// TIA Portal V20 export
FUNCTION_BLOCK "Sequence_1_Cutter"   // FB125, LAD
TITLE = Sequence
// Sequence template programmend in ladder logic
// stored: IsIECCheckEnabled true, MemoryReserve 100, Namespace Unit1.Em4, SetENOAutomatically true
   VAR
      instSequenceLADControl { ExternalWritable := 'False'} : "LAF_ControlLadSequence";
      instSequenceLADStatus { ExternalWritable := 'False'} : "LAF_StatusLadSequence";
      statPulse { ExternalWritable := 'False'} : Array[0..999] of Bool;
      statTonTimer { ExternalWritable := 'False'} : Array[0..999] of TON_TIME;
   END_VAR
   VAR_TEMP
      tempCustomerAction : Bool;   // Placeholder for possible actions
      tempDo_nothing_and_wait_for_init : Bool;   // Placeholder for doing nothing
      tempSafeStateCondition : Bool;   // Temp Condition for the equipment module to be in a safe state
   END_VAR
   VAR CONSTANT
      STEP_IDLE : DInt := 1;   // Idle Step
      JOB_1_STEP_01 : DInt := 101;
      JOB_1_STEP_11 : DInt := 111;
      JOB_1_STEP_21 : DInt := 121;
      JOB_1_STEP_31 : DInt := 131;
      JOB_1_STEP_41 : DInt := 141;
      JOB_1_STEP_51 : DInt := 151;
      JOB_1_STEP_61 : DInt := 161;
      JOB_1_STEP_71 : DInt := 171;
      JOB_1_STEP_81 : DInt := 181;
      JOB_1_STEP_91 : DInt := 191;
      JOB_2_STEP_01 : DInt := 201;
      JOB_2_STEP_11 : DInt := 211;
      JOB_2_STEP_21 : DInt := 221;
      JOB_2_STEP_31 : DInt := 231;
      JOB_2_STEP_41 : DInt := 241;
      JOB_2_STEP_51 : DInt := 251;
      JOB_2_STEP_61 : DInt := 261;
      JOB_2_STEP_71 : DInt := 271;
      JOB_2_STEP_81 : DInt := 281;
      JOB_2_STEP_91 : DInt := 291;
      JOB_3_STEP_01 : DInt := 301;
      JOB_3_STEP_11 : DInt := 311;
      JOB_3_STEP_21 : DInt := 321;
      JOB_3_STEP_31 : DInt := 331;
      JOB_3_STEP_41 : DInt := 341;
      JOB_3_STEP_51 : DInt := 351;
      JOB_3_STEP_61 : DInt := 361;
      JOB_3_STEP_71 : DInt := 371;
      JOB_3_STEP_81 : DInt := 381;
      JOB_3_STEP_91 : DInt := 391;
      JOB_4_STEP_01 : DInt := 401;
      JOB_4_STEP_11 : DInt := 411;
      JOB_4_STEP_21 : DInt := 421;
      JOB_4_STEP_31 : DInt := 431;
      JOB_4_STEP_41 : DInt := 441;
      JOB_4_STEP_51 : DInt := 451;
      JOB_4_STEP_61 : DInt := 461;
      JOB_4_STEP_71 : DInt := 471;
      JOB_4_STEP_81 : DInt := 481;
      JOB_4_STEP_91 : DInt := 491;
      STEP_IMMEDIATE_STOP : DInt := 901;   // Step executed when an immediate stop command is triggered for the sequence (i.e. when unit is in state aborting)
      SeqDelayTime : Time := T#100ms;
      SeqNoDelayTime : Time;
      TRUE : Bool := TRUE;
      FALSE : Bool := FALSE;
      PositionMovingAxisXCuttingPos : SInt := 1;
   END_VAR
   VAR_TEMP   // added for the SCL form of the ladder/FBD networks
      _w1 : Bool;
   END_VAR
BEGIN

REGION Network 1: BLOCK INFO HEADER
   // (company) / (C) Copyright (year)
   // ---------------------------------------------------------------------------------
   // Title:                             (Title of this block)
   // Comment/Function: (that is implemented in the block)
   // Library/Family:           (that the source is dedicated to)
   // Author:                        (department / person in charge / contact)
   // Target System:          (test system with FW version)
   // Engineering:              TIA Portal (SW version)
   // Restrictions:               (OB types, etc.)
   // Requirements:           (hardware, technological package, etc.)
   // ---------------------------------------------------------------------------------
   // Change log table:
   // Version          | Date             | Signature      | Expert in charge  | Changes applied ------------------------|----------------------|-------------------------|--------------------------------|-----------------------
   // 001.000.000 | yyyy-mm-dd | 0x00000000 | (name of expert) | First released version
END_REGION

REGION Network 2: DESCRIPTION
   // This is a template block provided by the Automation Framework. It can be used to create an own project.
   // The Block Info Header is prepared to put in your own data.
   // Description of the block could be added here and the docu created by Code2Docu.
END_REGION

REGION Network 3: ******************** CONTROL ********************
END_REGION

REGION Network 4: Sequence Control
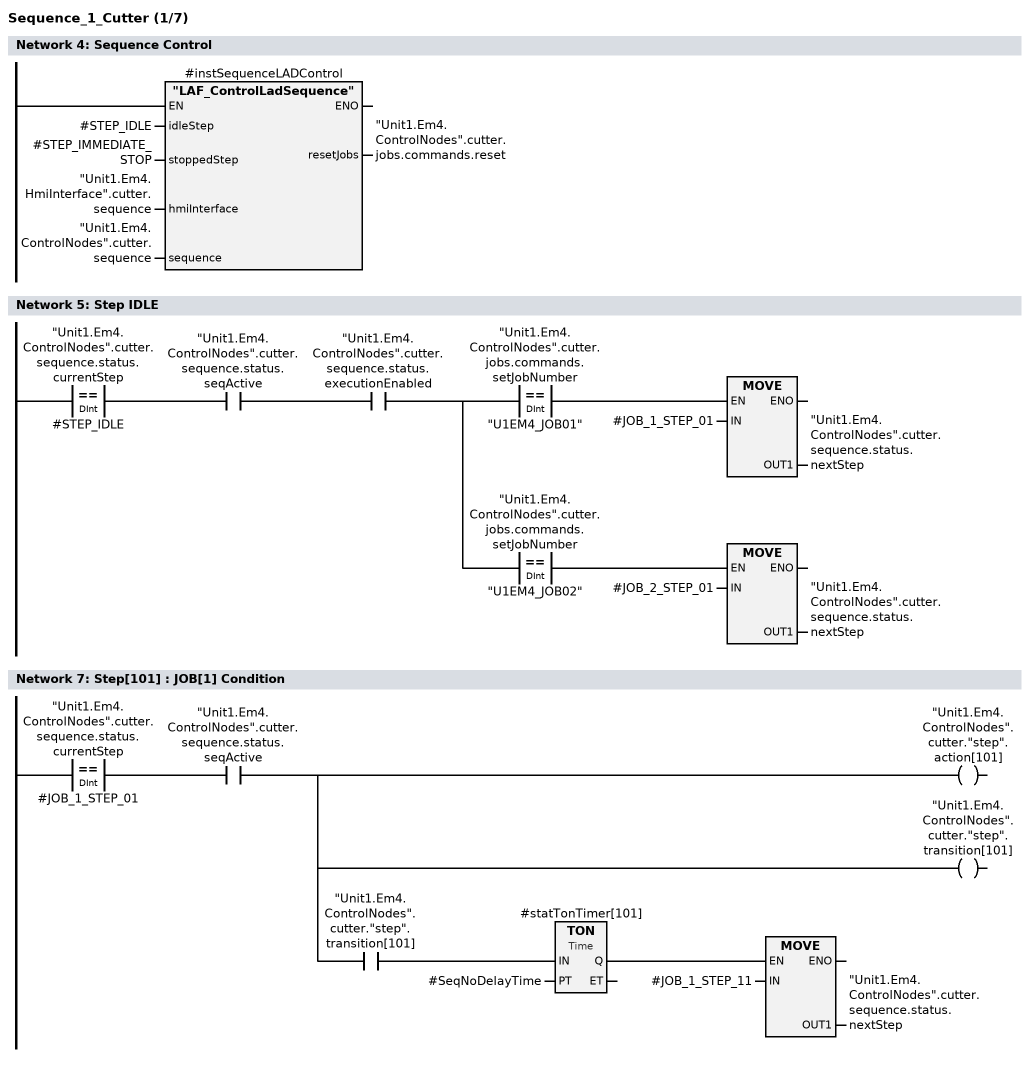
   RUNG wire#powerrail
      #instSequenceLADControl(idleStep := #STEP_IDLE, stoppedStep := #STEP_IMMEDIATE_STOP, hmiInterface := "Unit1.Em4.HmiInterface".cutter.sequence, sequence := "Unit1.Em4.ControlNodes".cutter.sequence, resetJobs => "Unit1.Em4.ControlNodes".cutter.jobs.commands.reset)
   END_RUNG
   // the same network as SCL:
   #instSequenceLADControl(idleStep := #STEP_IDLE,   // "LAF_ControlLadSequence"
                           stoppedStep := #STEP_IMMEDIATE_STOP,
                           hmiInterface := "Unit1.Em4.HmiInterface".cutter.sequence,
                           sequence := "Unit1.Em4.ControlNodes".cutter.sequence,
                           resetJobs => "Unit1.Em4.ControlNodes".cutter.jobs.commands.reset);
END_REGION

REGION Network 5: Step IDLE
   RUNG wire#powerrail
      { S7_Templates := "SrcType := DInt" } EQ_Contact(in1 := "Unit1.Em4.ControlNodes".cutter.sequence.status.currentStep, in2 := #STEP_IDLE)
      Contact( "Unit1.Em4.ControlNodes".cutter.sequence.status.seqActive )
      Contact( "Unit1.Em4.ControlNodes".cutter.sequence.status.executionEnabled )
      wire#w1
      { S7_Templates := "SrcType := DInt" } EQ_Contact(in1 := "Unit1.Em4.ControlNodes".cutter.jobs.commands.setJobNumber, in2 := "U1EM4_JOB01")
      Move(in := #JOB_1_STEP_01, out1 => "Unit1.Em4.ControlNodes".cutter.sequence.status.nextStep)
   END_RUNG
   RUNG wire#w1
      { S7_Templates := "SrcType := DInt" } EQ_Contact(in1 := "Unit1.Em4.ControlNodes".cutter.jobs.commands.setJobNumber, in2 := "U1EM4_JOB02")
      Move(in := #JOB_2_STEP_01, out1 => "Unit1.Em4.ControlNodes".cutter.sequence.status.nextStep)
   END_RUNG
   // the same network as SCL:
   #_w1 := ("Unit1.Em4.ControlNodes".cutter.sequence.status.currentStep = #STEP_IDLE) AND "Unit1.Em4.ControlNodes".cutter.sequence.status.seqActive AND "Unit1.Em4.ControlNodes".cutter.sequence.status.executionEnabled;
   IF #_w1 AND ("Unit1.Em4.ControlNodes".cutter.jobs.commands.setJobNumber = "U1EM4_JOB01") THEN
       "Unit1.Em4.ControlNodes".cutter.sequence.status.nextStep := #JOB_1_STEP_01;
   END_IF;
   IF #_w1 AND ("Unit1.Em4.ControlNodes".cutter.jobs.commands.setJobNumber = "U1EM4_JOB02") THEN
       "Unit1.Em4.ControlNodes".cutter.sequence.status.nextStep := #JOB_2_STEP_01;
   END_IF;
END_REGION

REGION Network 6: ******************** JOB[1] EM INITIALIZED ********************
END_REGION

REGION Network 7: Step[101] : JOB[1] Condition
   RUNG wire#powerrail
      { S7_Templates := "SrcType := DInt" } EQ_Contact(in1 := "Unit1.Em4.ControlNodes".cutter.sequence.status.currentStep, in2 := #JOB_1_STEP_01)
      Contact( "Unit1.Em4.ControlNodes".cutter.sequence.status.seqActive )
      wire#w1
      Coil( "Unit1.Em4.ControlNodes".cutter."step".action[101] )
   END_RUNG
   RUNG wire#w1
      Coil( "Unit1.Em4.ControlNodes".cutter."step".transition[101] )
   END_RUNG
   RUNG wire#w1
      Contact( "Unit1.Em4.ControlNodes".cutter."step".transition[101] )
      { S7_Templates := "time_type := Time" } #statTonTimer[101].TON(pt := #SeqNoDelayTime, et =>)
      Move(in := #JOB_1_STEP_11, out1 => "Unit1.Em4.ControlNodes".cutter.sequence.status.nextStep)
   END_RUNG
   // the same network as SCL:
   "Unit1.Em4.ControlNodes".cutter."step".action[101] := ("Unit1.Em4.ControlNodes".cutter.sequence.status.currentStep = #JOB_1_STEP_01) AND "Unit1.Em4.ControlNodes".cutter.sequence.status.seqActive;
   "Unit1.Em4.ControlNodes".cutter."step".transition[101] := ("Unit1.Em4.ControlNodes".cutter.sequence.status.currentStep = #JOB_1_STEP_01) AND "Unit1.Em4.ControlNodes".cutter.sequence.status.seqActive;
   #statTonTimer[101].TON(IN := ("Unit1.Em4.ControlNodes".cutter.sequence.status.currentStep = #JOB_1_STEP_01) AND "Unit1.Em4.ControlNodes".cutter.sequence.status.seqActive AND "Unit1.Em4.ControlNodes".cutter."step".transition[101],
                          PT := #SeqNoDelayTime);
   IF #statTonTimer[101].Q THEN
       "Unit1.Em4.ControlNodes".cutter.sequence.status.nextStep := #JOB_1_STEP_11;
   END_IF;
END_REGION

REGION Network 8: Step[111] : Axis Homed Check
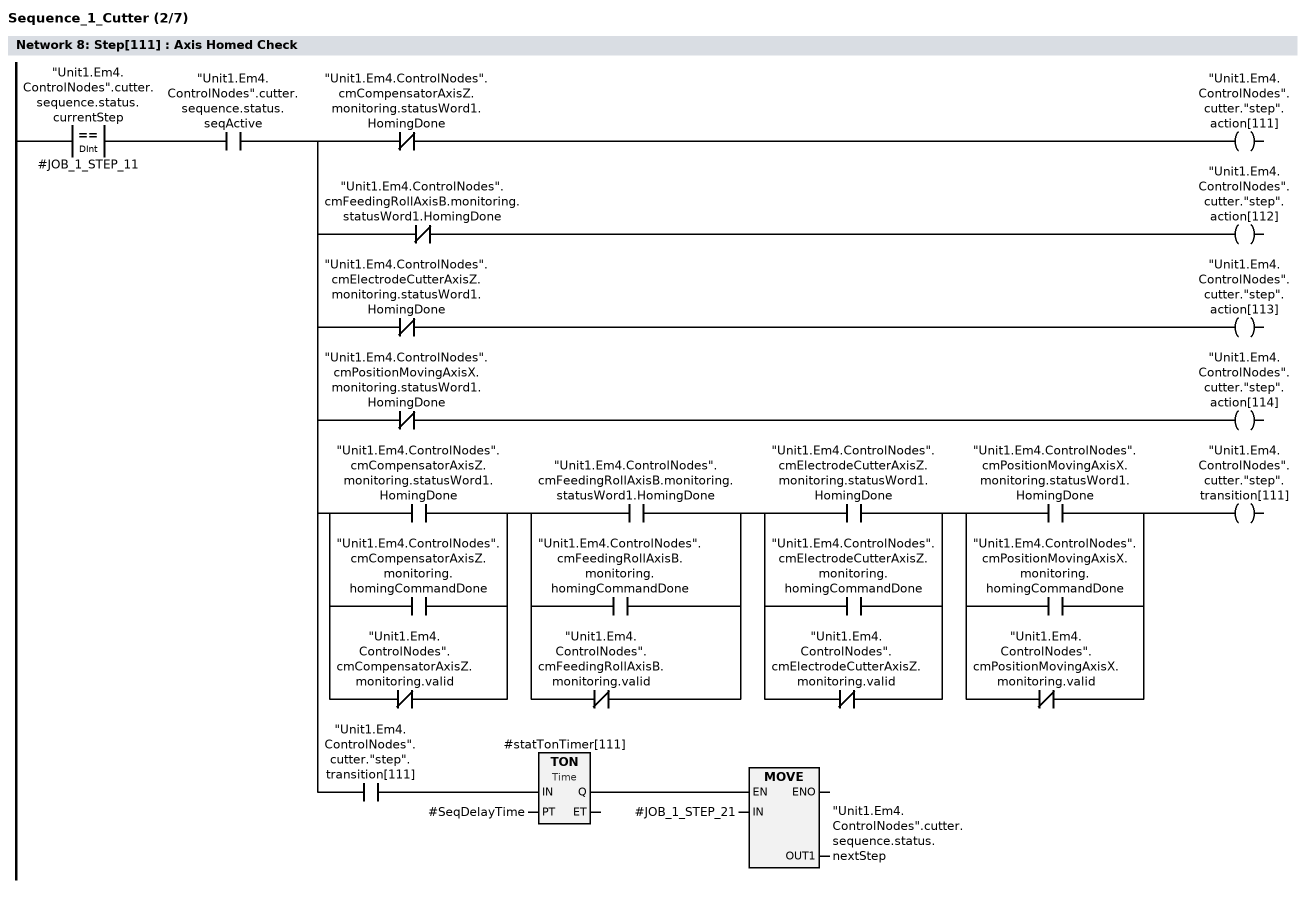
   RUNG wire#powerrail
      { S7_Templates := "SrcType := DInt" } EQ_Contact(in1 := "Unit1.Em4.ControlNodes".cutter.sequence.status.currentStep, in2 := #JOB_1_STEP_11)
      Contact( "Unit1.Em4.ControlNodes".cutter.sequence.status.seqActive )
      wire#w1
      I_Contact( "Unit1.Em4.ControlNodes".cmCompensatorAxisZ.monitoring.statusWord1.HomingDone )
      Coil( "Unit1.Em4.ControlNodes".cutter."step".action[111] )
   END_RUNG
   RUNG wire#w1
      I_Contact( "Unit1.Em4.ControlNodes".cmFeedingRollAxisB.monitoring.statusWord1.HomingDone )
      Coil( "Unit1.Em4.ControlNodes".cutter."step".action[112] )
   END_RUNG
   RUNG wire#w1
      I_Contact( "Unit1.Em4.ControlNodes".cmElectrodeCutterAxisZ.monitoring.statusWord1.HomingDone )
      Coil( "Unit1.Em4.ControlNodes".cutter."step".action[113] )
   END_RUNG
   RUNG wire#w1
      I_Contact( "Unit1.Em4.ControlNodes".cmPositionMovingAxisX.monitoring.statusWord1.HomingDone )
      Coil( "Unit1.Em4.ControlNodes".cutter."step".action[114] )
   END_RUNG
   RUNG wire#w1
      Contact( "Unit1.Em4.ControlNodes".cmCompensatorAxisZ.monitoring.statusWord1.HomingDone )
      wire#w2
      Contact( "Unit1.Em4.ControlNodes".cmFeedingRollAxisB.monitoring.statusWord1.HomingDone )
      wire#w3
      Contact( "Unit1.Em4.ControlNodes".cmElectrodeCutterAxisZ.monitoring.statusWord1.HomingDone )
      wire#w4
      Contact( "Unit1.Em4.ControlNodes".cmPositionMovingAxisX.monitoring.statusWord1.HomingDone )
      wire#w5
      Coil( "Unit1.Em4.ControlNodes".cutter."step".transition[111] )
   END_RUNG
   RUNG wire#w1
      Contact( "Unit1.Em4.ControlNodes".cmCompensatorAxisZ.monitoring.homingCommandDone )
   END_RUNG wire#w2
   RUNG wire#w1
      I_Contact( "Unit1.Em4.ControlNodes".cmCompensatorAxisZ.monitoring.valid )
   END_RUNG wire#w2
   RUNG wire#w2
      Contact( "Unit1.Em4.ControlNodes".cmFeedingRollAxisB.monitoring.homingCommandDone )
   END_RUNG wire#w3
   RUNG wire#w2
      I_Contact( "Unit1.Em4.ControlNodes".cmFeedingRollAxisB.monitoring.valid )
   END_RUNG wire#w3
   RUNG wire#w3
      Contact( "Unit1.Em4.ControlNodes".cmElectrodeCutterAxisZ.monitoring.homingCommandDone )
   END_RUNG wire#w4
   RUNG wire#w3
      I_Contact( "Unit1.Em4.ControlNodes".cmElectrodeCutterAxisZ.monitoring.valid )
   END_RUNG wire#w4
   RUNG wire#w4
      Contact( "Unit1.Em4.ControlNodes".cmPositionMovingAxisX.monitoring.homingCommandDone )
   END_RUNG wire#w5
   RUNG wire#w4
      I_Contact( "Unit1.Em4.ControlNodes".cmPositionMovingAxisX.monitoring.valid )
   END_RUNG wire#w5
   RUNG wire#w1
      Contact( "Unit1.Em4.ControlNodes".cutter."step".transition[111] )
      { S7_Templates := "time_type := Time" } #statTonTimer[111].TON(pt := #SeqDelayTime, et =>)
      Move(in := #JOB_1_STEP_21, out1 => "Unit1.Em4.ControlNodes".cutter.sequence.status.nextStep)
   END_RUNG
   // the same network as SCL:
   #_w1 := ("Unit1.Em4.ControlNodes".cutter.sequence.status.currentStep = #JOB_1_STEP_11) AND "Unit1.Em4.ControlNodes".cutter.sequence.status.seqActive;
   "Unit1.Em4.ControlNodes".cutter."step".action[111] := #_w1 AND NOT "Unit1.Em4.ControlNodes".cmCompensatorAxisZ.monitoring.statusWord1.HomingDone;
   "Unit1.Em4.ControlNodes".cutter."step".action[112] := #_w1 AND NOT "Unit1.Em4.ControlNodes".cmFeedingRollAxisB.monitoring.statusWord1.HomingDone;
   "Unit1.Em4.ControlNodes".cutter."step".action[113] := #_w1 AND NOT "Unit1.Em4.ControlNodes".cmElectrodeCutterAxisZ.monitoring.statusWord1.HomingDone;
   "Unit1.Em4.ControlNodes".cutter."step".action[114] := #_w1 AND NOT "Unit1.Em4.ControlNodes".cmPositionMovingAxisX.monitoring.statusWord1.HomingDone;
   "Unit1.Em4.ControlNodes".cutter."step".transition[111] := #_w1 AND ("Unit1.Em4.ControlNodes".cmCompensatorAxisZ.monitoring.statusWord1.HomingDone OR "Unit1.Em4.ControlNodes".cmCompensatorAxisZ.monitoring.homingCommandDone OR NOT "Unit1.Em4.ControlNodes".cmCompensatorAxisZ.monitoring.valid) AND ("Unit1.Em4.ControlNodes".cmFeedingRollAxisB.monitoring.statusWord1.HomingDone OR "Unit1.Em4.ControlNodes".cmFeedingRollAxisB.monitoring.homingCommandDone OR NOT "Unit1.Em4.ControlNodes".cmFeedingRollAxisB.monitoring.valid) AND ("Unit1.Em4.ControlNodes".cmElectrodeCutterAxisZ.monitoring.statusWord1.HomingDone OR "Unit1.Em4.ControlNodes".cmElectrodeCutterAxisZ.monitoring.homingCommandDone OR NOT "Unit1.Em4.ControlNodes".cmElectrodeCutterAxisZ.monitoring.valid) AND ("Unit1.Em4.ControlNodes".cmPositionMovingAxisX.monitoring.statusWord1.HomingDone OR "Unit1.Em4.ControlNodes".cmPositionMovingAxisX.monitoring.homingCommandDone OR NOT "Unit1.Em4.ControlNodes".cmPositionMovingAxisX.monitoring.valid);
   #statTonTimer[111].TON(IN := #_w1 AND "Unit1.Em4.ControlNodes".cutter."step".transition[111],
                          PT := #SeqDelayTime);
   IF #statTonTimer[111].Q THEN
       "Unit1.Em4.ControlNodes".cutter.sequence.status.nextStep := #JOB_1_STEP_21;
   END_IF;
END_REGION

REGION Network 9: Step[121] : Axis HomePos Check
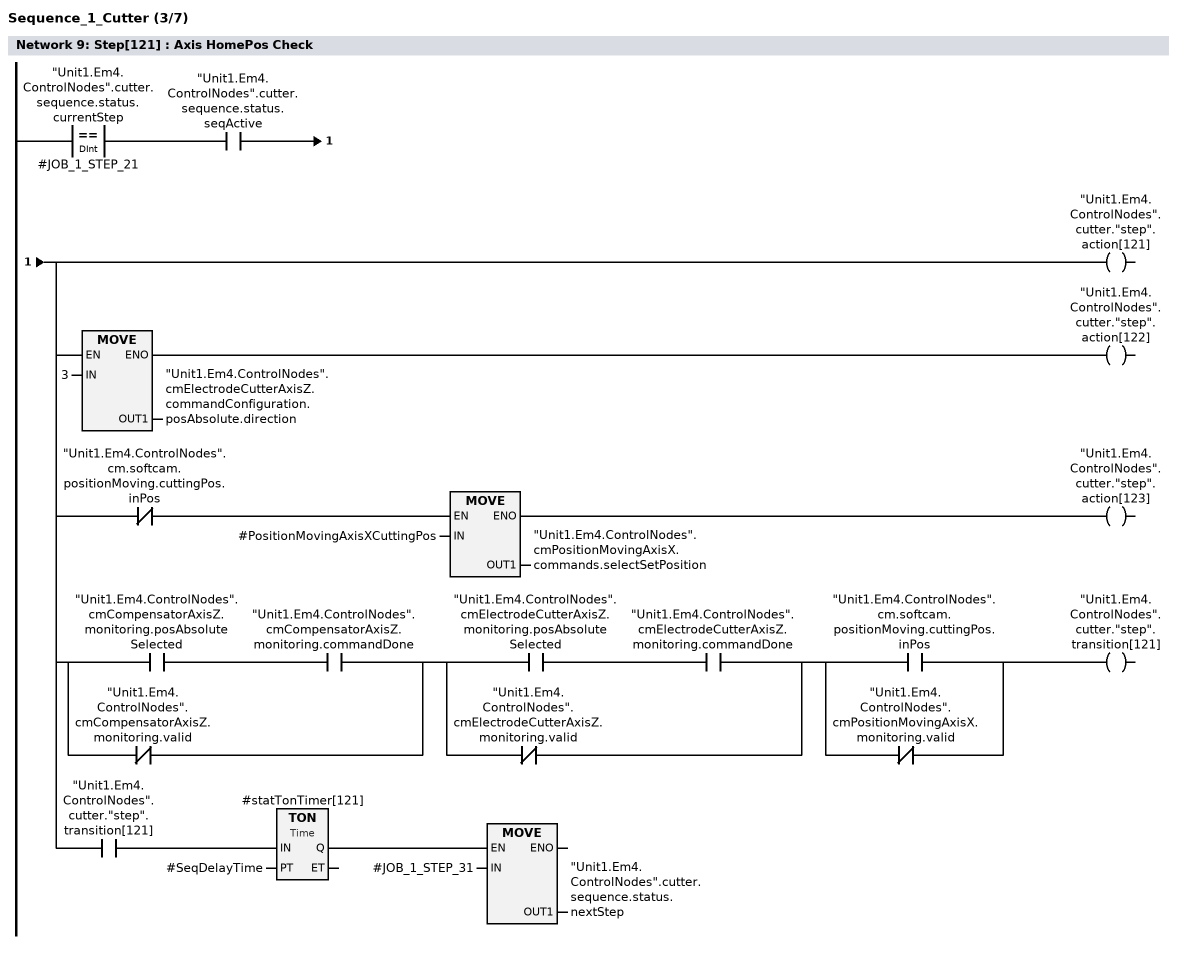
   RUNG wire#powerrail
      { S7_Templates := "SrcType := DInt" } EQ_Contact(in1 := "Unit1.Em4.ControlNodes".cutter.sequence.status.currentStep, in2 := #JOB_1_STEP_21)
      Contact( "Unit1.Em4.ControlNodes".cutter.sequence.status.seqActive )
      wire#w1
      Coil( "Unit1.Em4.ControlNodes".cutter."step".action[121] )
   END_RUNG
   RUNG wire#w1
      Move(in := 3, out1 => "Unit1.Em4.ControlNodes".cmElectrodeCutterAxisZ.commandConfiguration.posAbsolute.direction)
      Coil( "Unit1.Em4.ControlNodes".cutter."step".action[122] )
   END_RUNG
   RUNG wire#w1
      I_Contact( "Unit1.Em4.ControlNodes".cm.softcam.positionMoving.cuttingPos.inPos )
      Move(in := #PositionMovingAxisXCuttingPos, out1 => "Unit1.Em4.ControlNodes".cmPositionMovingAxisX.commands.selectSetPosition)
      Coil( "Unit1.Em4.ControlNodes".cutter."step".action[123] )
   END_RUNG
   RUNG wire#w1
      Contact( "Unit1.Em4.ControlNodes".cmCompensatorAxisZ.monitoring.posAbsoluteSelected )
      Contact( "Unit1.Em4.ControlNodes".cmCompensatorAxisZ.monitoring.commandDone )
      wire#w2
      Contact( "Unit1.Em4.ControlNodes".cmElectrodeCutterAxisZ.monitoring.posAbsoluteSelected )
      Contact( "Unit1.Em4.ControlNodes".cmElectrodeCutterAxisZ.monitoring.commandDone )
      wire#w3
      Contact( "Unit1.Em4.ControlNodes".cm.softcam.positionMoving.cuttingPos.inPos )
      wire#w4
      Coil( "Unit1.Em4.ControlNodes".cutter."step".transition[121] )
   END_RUNG
   RUNG wire#w1
      I_Contact( "Unit1.Em4.ControlNodes".cmCompensatorAxisZ.monitoring.valid )
   END_RUNG wire#w2
   RUNG wire#w2
      I_Contact( "Unit1.Em4.ControlNodes".cmElectrodeCutterAxisZ.monitoring.valid )
   END_RUNG wire#w3
   RUNG wire#w3
      I_Contact( "Unit1.Em4.ControlNodes".cmPositionMovingAxisX.monitoring.valid )
   END_RUNG wire#w4
   RUNG wire#w1
      Contact( "Unit1.Em4.ControlNodes".cutter."step".transition[121] )
      { S7_Templates := "time_type := Time" } #statTonTimer[121].TON(pt := #SeqDelayTime, et =>)
      Move(in := #JOB_1_STEP_31, out1 => "Unit1.Em4.ControlNodes".cutter.sequence.status.nextStep)
   END_RUNG
   // the same network as SCL:
   "Unit1.Em4.ControlNodes".cutter."step".action[121] := ("Unit1.Em4.ControlNodes".cutter.sequence.status.currentStep = #JOB_1_STEP_21) AND "Unit1.Em4.ControlNodes".cutter.sequence.status.seqActive;
   IF ("Unit1.Em4.ControlNodes".cutter.sequence.status.currentStep = #JOB_1_STEP_21) AND "Unit1.Em4.ControlNodes".cutter.sequence.status.seqActive THEN
       "Unit1.Em4.ControlNodes".cmElectrodeCutterAxisZ.commandConfiguration.posAbsolute.direction := 3;
   END_IF;
   "Unit1.Em4.ControlNodes".cutter."step".action[122] := ("Unit1.Em4.ControlNodes".cutter.sequence.status.currentStep = #JOB_1_STEP_21) AND "Unit1.Em4.ControlNodes".cutter.sequence.status.seqActive;
   #_w1 := ("Unit1.Em4.ControlNodes".cutter.sequence.status.currentStep = #JOB_1_STEP_21) AND "Unit1.Em4.ControlNodes".cutter.sequence.status.seqActive AND NOT "Unit1.Em4.ControlNodes".cm.softcam.positionMoving.cuttingPos.inPos;
   IF #_w1 THEN
       "Unit1.Em4.ControlNodes".cmPositionMovingAxisX.commands.selectSetPosition := #PositionMovingAxisXCuttingPos;
   END_IF;
   "Unit1.Em4.ControlNodes".cutter."step".action[123] := #_w1;
   "Unit1.Em4.ControlNodes".cutter."step".transition[121] := ("Unit1.Em4.ControlNodes".cutter.sequence.status.currentStep = #JOB_1_STEP_21) AND "Unit1.Em4.ControlNodes".cutter.sequence.status.seqActive AND (("Unit1.Em4.ControlNodes".cmCompensatorAxisZ.monitoring.posAbsoluteSelected AND "Unit1.Em4.ControlNodes".cmCompensatorAxisZ.monitoring.commandDone) OR NOT "Unit1.Em4.ControlNodes".cmCompensatorAxisZ.monitoring.valid) AND (("Unit1.Em4.ControlNodes".cmElectrodeCutterAxisZ.monitoring.posAbsoluteSelected AND "Unit1.Em4.ControlNodes".cmElectrodeCutterAxisZ.monitoring.commandDone) OR NOT "Unit1.Em4.ControlNodes".cmElectrodeCutterAxisZ.monitoring.valid) AND ("Unit1.Em4.ControlNodes".cm.softcam.positionMoving.cuttingPos.inPos OR NOT "Unit1.Em4.ControlNodes".cmPositionMovingAxisX.monitoring.valid);
   #statTonTimer[121].TON(IN := ("Unit1.Em4.ControlNodes".cutter.sequence.status.currentStep = #JOB_1_STEP_21) AND "Unit1.Em4.ControlNodes".cutter.sequence.status.seqActive AND "Unit1.Em4.ControlNodes".cutter."step".transition[121],
                          PT := #SeqDelayTime);
   IF #statTonTimer[121].Q THEN
       "Unit1.Em4.ControlNodes".cutter.sequence.status.nextStep := #JOB_1_STEP_31;
   END_IF;
END_REGION

REGION Network 10: Step[131] : Feeding Cylinder WorkPos Check
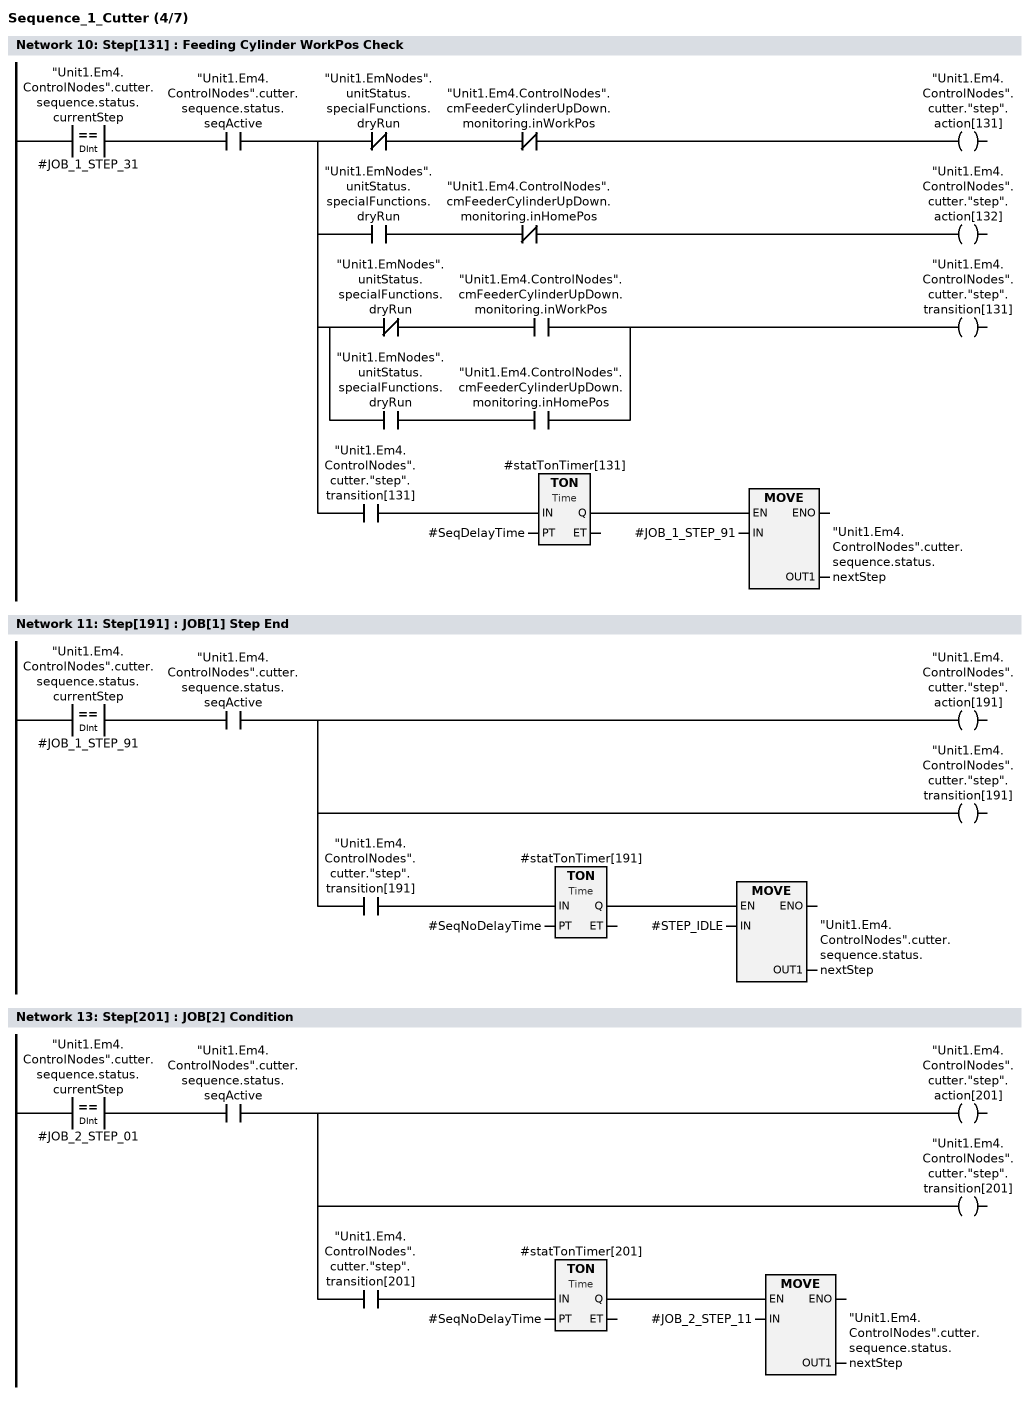
   RUNG wire#powerrail
      { S7_Templates := "SrcType := DInt" } EQ_Contact(in1 := "Unit1.Em4.ControlNodes".cutter.sequence.status.currentStep, in2 := #JOB_1_STEP_31)
      Contact( "Unit1.Em4.ControlNodes".cutter.sequence.status.seqActive )
      wire#w1
      I_Contact( "Unit1.EmNodes".unitStatus.specialFunctions.dryRun )
      I_Contact( "Unit1.Em4.ControlNodes".cmFeederCylinderUpDown.monitoring.inWorkPos )
      Coil( "Unit1.Em4.ControlNodes".cutter."step".action[131] )
   END_RUNG
   RUNG wire#w1
      Contact( "Unit1.EmNodes".unitStatus.specialFunctions.dryRun )
      I_Contact( "Unit1.Em4.ControlNodes".cmFeederCylinderUpDown.monitoring.inHomePos )
      Coil( "Unit1.Em4.ControlNodes".cutter."step".action[132] )
   END_RUNG
   RUNG wire#w1
      I_Contact( "Unit1.EmNodes".unitStatus.specialFunctions.dryRun )
      Contact( "Unit1.Em4.ControlNodes".cmFeederCylinderUpDown.monitoring.inWorkPos )
      wire#w2
      Coil( "Unit1.Em4.ControlNodes".cutter."step".transition[131] )
   END_RUNG
   RUNG wire#w1
      Contact( "Unit1.EmNodes".unitStatus.specialFunctions.dryRun )
      Contact( "Unit1.Em4.ControlNodes".cmFeederCylinderUpDown.monitoring.inHomePos )
   END_RUNG wire#w2
   RUNG wire#w1
      Contact( "Unit1.Em4.ControlNodes".cutter."step".transition[131] )
      { S7_Templates := "time_type := Time" } #statTonTimer[131].TON(pt := #SeqDelayTime, et =>)
      Move(in := #JOB_1_STEP_91, out1 => "Unit1.Em4.ControlNodes".cutter.sequence.status.nextStep)
   END_RUNG
   // the same network as SCL:
   #_w1 := ("Unit1.Em4.ControlNodes".cutter.sequence.status.currentStep = #JOB_1_STEP_31) AND "Unit1.Em4.ControlNodes".cutter.sequence.status.seqActive;
   "Unit1.Em4.ControlNodes".cutter."step".action[131] := #_w1 AND NOT "Unit1.EmNodes".unitStatus.specialFunctions.dryRun AND NOT "Unit1.Em4.ControlNodes".cmFeederCylinderUpDown.monitoring.inWorkPos;
   "Unit1.Em4.ControlNodes".cutter."step".action[132] := #_w1 AND "Unit1.EmNodes".unitStatus.specialFunctions.dryRun AND NOT "Unit1.Em4.ControlNodes".cmFeederCylinderUpDown.monitoring.inHomePos;
   "Unit1.Em4.ControlNodes".cutter."step".transition[131] := #_w1 AND ((NOT "Unit1.EmNodes".unitStatus.specialFunctions.dryRun AND "Unit1.Em4.ControlNodes".cmFeederCylinderUpDown.monitoring.inWorkPos) OR ("Unit1.EmNodes".unitStatus.specialFunctions.dryRun AND "Unit1.Em4.ControlNodes".cmFeederCylinderUpDown.monitoring.inHomePos));
   #statTonTimer[131].TON(IN := #_w1 AND "Unit1.Em4.ControlNodes".cutter."step".transition[131],
                          PT := #SeqDelayTime);
   IF #statTonTimer[131].Q THEN
       "Unit1.Em4.ControlNodes".cutter.sequence.status.nextStep := #JOB_1_STEP_91;
   END_IF;
END_REGION

REGION Network 11: Step[191] : JOB[1] Step End
   RUNG wire#powerrail
      { S7_Templates := "SrcType := DInt" } EQ_Contact(in1 := "Unit1.Em4.ControlNodes".cutter.sequence.status.currentStep, in2 := #JOB_1_STEP_91)
      Contact( "Unit1.Em4.ControlNodes".cutter.sequence.status.seqActive )
      wire#w1
      Coil( "Unit1.Em4.ControlNodes".cutter."step".action[191] )
   END_RUNG
   RUNG wire#w1
      Coil( "Unit1.Em4.ControlNodes".cutter."step".transition[191] )
   END_RUNG
   RUNG wire#w1
      Contact( "Unit1.Em4.ControlNodes".cutter."step".transition[191] )
      { S7_Templates := "time_type := Time" } #statTonTimer[191].TON(pt := #SeqNoDelayTime, et =>)
      Move(in := #STEP_IDLE, out1 => "Unit1.Em4.ControlNodes".cutter.sequence.status.nextStep)
   END_RUNG
   // the same network as SCL:
   "Unit1.Em4.ControlNodes".cutter."step".action[191] := ("Unit1.Em4.ControlNodes".cutter.sequence.status.currentStep = #JOB_1_STEP_91) AND "Unit1.Em4.ControlNodes".cutter.sequence.status.seqActive;
   "Unit1.Em4.ControlNodes".cutter."step".transition[191] := ("Unit1.Em4.ControlNodes".cutter.sequence.status.currentStep = #JOB_1_STEP_91) AND "Unit1.Em4.ControlNodes".cutter.sequence.status.seqActive;
   #statTonTimer[191].TON(IN := ("Unit1.Em4.ControlNodes".cutter.sequence.status.currentStep = #JOB_1_STEP_91) AND "Unit1.Em4.ControlNodes".cutter.sequence.status.seqActive AND "Unit1.Em4.ControlNodes".cutter."step".transition[191],
                          PT := #SeqNoDelayTime);
   IF #statTonTimer[191].Q THEN
       "Unit1.Em4.ControlNodes".cutter.sequence.status.nextStep := #STEP_IDLE;
   END_IF;
END_REGION

REGION Network 12: ******************** JOB[2] Cutter One Cycle ********************
END_REGION

REGION Network 13: Step[201] : JOB[2] Condition
   RUNG wire#powerrail
      { S7_Templates := "SrcType := DInt" } EQ_Contact(in1 := "Unit1.Em4.ControlNodes".cutter.sequence.status.currentStep, in2 := #JOB_2_STEP_01)
      Contact( "Unit1.Em4.ControlNodes".cutter.sequence.status.seqActive )
      wire#w1
      Coil( "Unit1.Em4.ControlNodes".cutter."step".action[201] )
   END_RUNG
   RUNG wire#w1
      Coil( "Unit1.Em4.ControlNodes".cutter."step".transition[201] )
   END_RUNG
   RUNG wire#w1
      Contact( "Unit1.Em4.ControlNodes".cutter."step".transition[201] )
      { S7_Templates := "time_type := Time" } #statTonTimer[201].TON(pt := #SeqNoDelayTime, et =>)
      Move(in := #JOB_2_STEP_11, out1 => "Unit1.Em4.ControlNodes".cutter.sequence.status.nextStep)
   END_RUNG
   // the same network as SCL:
   "Unit1.Em4.ControlNodes".cutter."step".action[201] := ("Unit1.Em4.ControlNodes".cutter.sequence.status.currentStep = #JOB_2_STEP_01) AND "Unit1.Em4.ControlNodes".cutter.sequence.status.seqActive;
   "Unit1.Em4.ControlNodes".cutter."step".transition[201] := ("Unit1.Em4.ControlNodes".cutter.sequence.status.currentStep = #JOB_2_STEP_01) AND "Unit1.Em4.ControlNodes".cutter.sequence.status.seqActive;
   #statTonTimer[201].TON(IN := ("Unit1.Em4.ControlNodes".cutter.sequence.status.currentStep = #JOB_2_STEP_01) AND "Unit1.Em4.ControlNodes".cutter.sequence.status.seqActive AND "Unit1.Em4.ControlNodes".cutter."step".transition[201],
                          PT := #SeqNoDelayTime);
   IF #statTonTimer[201].Q THEN
       "Unit1.Em4.ControlNodes".cutter.sequence.status.nextStep := #JOB_2_STEP_11;
   END_IF;
END_REGION

REGION Network 14: Step[211] : Cutter Work Position
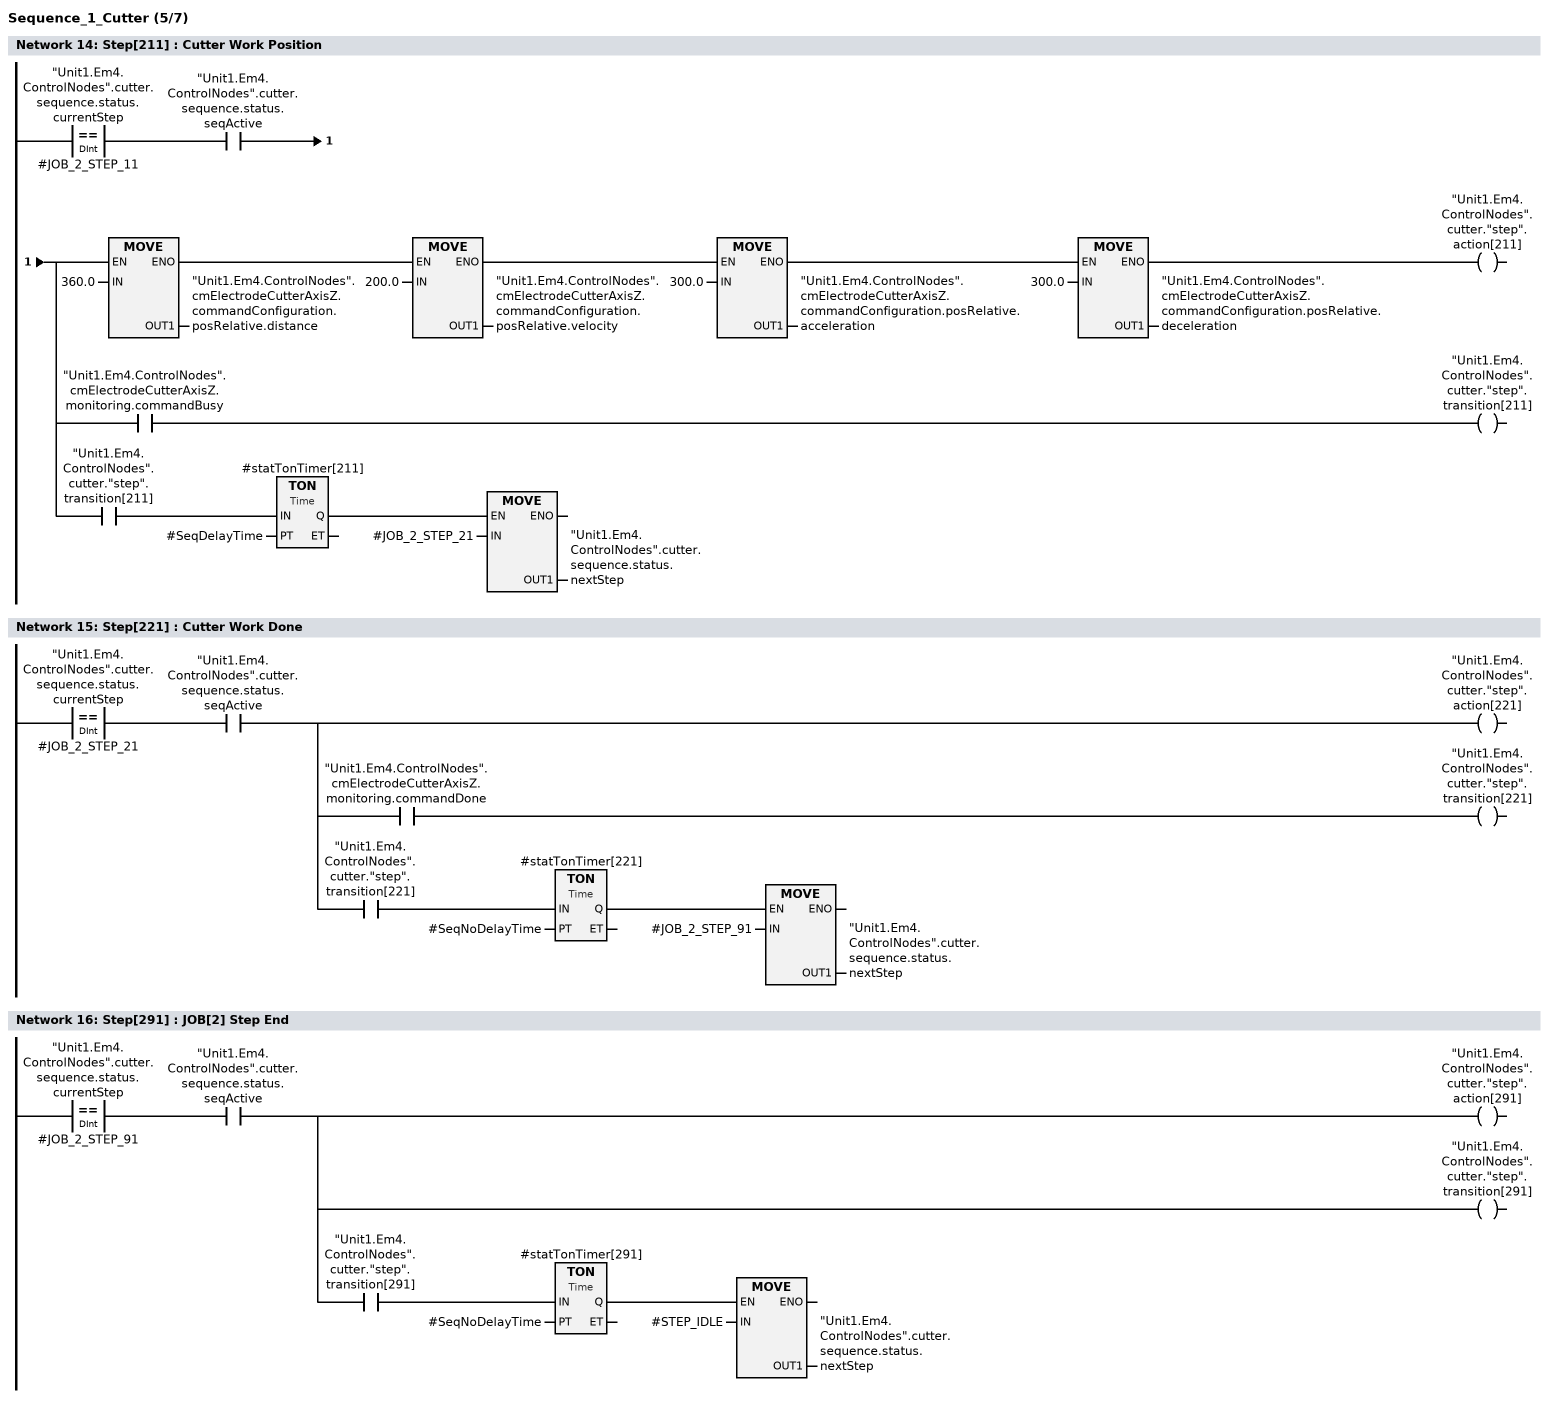
   RUNG wire#powerrail
      { S7_Templates := "SrcType := DInt" } EQ_Contact(in1 := "Unit1.Em4.ControlNodes".cutter.sequence.status.currentStep, in2 := #JOB_2_STEP_11)
      Contact( "Unit1.Em4.ControlNodes".cutter.sequence.status.seqActive )
      wire#w1
      Move(in := 360.0, out1 => "Unit1.Em4.ControlNodes".cmElectrodeCutterAxisZ.commandConfiguration.posRelative.distance)
      Move(in := 200.0, out1 => "Unit1.Em4.ControlNodes".cmElectrodeCutterAxisZ.commandConfiguration.posRelative.velocity)
      Move(in := 300.0, out1 => "Unit1.Em4.ControlNodes".cmElectrodeCutterAxisZ.commandConfiguration.posRelative.acceleration)
      Move(in := 300.0, out1 => "Unit1.Em4.ControlNodes".cmElectrodeCutterAxisZ.commandConfiguration.posRelative.deceleration)
      Coil( "Unit1.Em4.ControlNodes".cutter."step".action[211] )
   END_RUNG
   RUNG wire#w1
      Contact( "Unit1.Em4.ControlNodes".cmElectrodeCutterAxisZ.monitoring.commandBusy )
      Coil( "Unit1.Em4.ControlNodes".cutter."step".transition[211] )
   END_RUNG
   RUNG wire#w1
      Contact( "Unit1.Em4.ControlNodes".cutter."step".transition[211] )
      { S7_Templates := "time_type := Time" } #statTonTimer[211].TON(pt := #SeqDelayTime, et =>)
      Move(in := #JOB_2_STEP_21, out1 => "Unit1.Em4.ControlNodes".cutter.sequence.status.nextStep)
   END_RUNG
   // the same network as SCL:
   #_w1 := ("Unit1.Em4.ControlNodes".cutter.sequence.status.currentStep = #JOB_2_STEP_11) AND "Unit1.Em4.ControlNodes".cutter.sequence.status.seqActive;
   IF #_w1 THEN
       "Unit1.Em4.ControlNodes".cmElectrodeCutterAxisZ.commandConfiguration.posRelative.distance := 360.0;
       "Unit1.Em4.ControlNodes".cmElectrodeCutterAxisZ.commandConfiguration.posRelative.velocity := 200.0;
       "Unit1.Em4.ControlNodes".cmElectrodeCutterAxisZ.commandConfiguration.posRelative.acceleration := 300.0;
       "Unit1.Em4.ControlNodes".cmElectrodeCutterAxisZ.commandConfiguration.posRelative.deceleration := 300.0;
   END_IF;
   "Unit1.Em4.ControlNodes".cutter."step".action[211] := #_w1;
   "Unit1.Em4.ControlNodes".cutter."step".transition[211] := #_w1 AND "Unit1.Em4.ControlNodes".cmElectrodeCutterAxisZ.monitoring.commandBusy;
   #statTonTimer[211].TON(IN := #_w1 AND "Unit1.Em4.ControlNodes".cutter."step".transition[211],
                          PT := #SeqDelayTime);
   IF #statTonTimer[211].Q THEN
       "Unit1.Em4.ControlNodes".cutter.sequence.status.nextStep := #JOB_2_STEP_21;
   END_IF;
END_REGION

REGION Network 15: Step[221] : Cutter Work Done
   RUNG wire#powerrail
      { S7_Templates := "SrcType := DInt" } EQ_Contact(in1 := "Unit1.Em4.ControlNodes".cutter.sequence.status.currentStep, in2 := #JOB_2_STEP_21)
      Contact( "Unit1.Em4.ControlNodes".cutter.sequence.status.seqActive )
      wire#w1
      Coil( "Unit1.Em4.ControlNodes".cutter."step".action[221] )
   END_RUNG
   RUNG wire#w1
      Contact( "Unit1.Em4.ControlNodes".cmElectrodeCutterAxisZ.monitoring.commandDone )
      Coil( "Unit1.Em4.ControlNodes".cutter."step".transition[221] )
   END_RUNG
   RUNG wire#w1
      Contact( "Unit1.Em4.ControlNodes".cutter."step".transition[221] )
      { S7_Templates := "time_type := Time" } #statTonTimer[221].TON(pt := #SeqNoDelayTime, et =>)
      Move(in := #JOB_2_STEP_91, out1 => "Unit1.Em4.ControlNodes".cutter.sequence.status.nextStep)
   END_RUNG
   // the same network as SCL:
   "Unit1.Em4.ControlNodes".cutter."step".action[221] := ("Unit1.Em4.ControlNodes".cutter.sequence.status.currentStep = #JOB_2_STEP_21) AND "Unit1.Em4.ControlNodes".cutter.sequence.status.seqActive;
   "Unit1.Em4.ControlNodes".cutter."step".transition[221] := ("Unit1.Em4.ControlNodes".cutter.sequence.status.currentStep = #JOB_2_STEP_21) AND "Unit1.Em4.ControlNodes".cutter.sequence.status.seqActive AND "Unit1.Em4.ControlNodes".cmElectrodeCutterAxisZ.monitoring.commandDone;
   #statTonTimer[221].TON(IN := ("Unit1.Em4.ControlNodes".cutter.sequence.status.currentStep = #JOB_2_STEP_21) AND "Unit1.Em4.ControlNodes".cutter.sequence.status.seqActive AND "Unit1.Em4.ControlNodes".cutter."step".transition[221],
                          PT := #SeqNoDelayTime);
   IF #statTonTimer[221].Q THEN
       "Unit1.Em4.ControlNodes".cutter.sequence.status.nextStep := #JOB_2_STEP_91;
   END_IF;
END_REGION

REGION Network 16: Step[291] : JOB[2] Step End
   RUNG wire#powerrail
      { S7_Templates := "SrcType := DInt" } EQ_Contact(in1 := "Unit1.Em4.ControlNodes".cutter.sequence.status.currentStep, in2 := #JOB_2_STEP_91)
      Contact( "Unit1.Em4.ControlNodes".cutter.sequence.status.seqActive )
      wire#w1
      Coil( "Unit1.Em4.ControlNodes".cutter."step".action[291] )
   END_RUNG
   RUNG wire#w1
      Coil( "Unit1.Em4.ControlNodes".cutter."step".transition[291] )
   END_RUNG
   RUNG wire#w1
      Contact( "Unit1.Em4.ControlNodes".cutter."step".transition[291] )
      { S7_Templates := "time_type := Time" } #statTonTimer[291].TON(pt := #SeqNoDelayTime, et =>)
      Move(in := #STEP_IDLE, out1 => "Unit1.Em4.ControlNodes".cutter.sequence.status.nextStep)
   END_RUNG
   // the same network as SCL:
   "Unit1.Em4.ControlNodes".cutter."step".action[291] := ("Unit1.Em4.ControlNodes".cutter.sequence.status.currentStep = #JOB_2_STEP_91) AND "Unit1.Em4.ControlNodes".cutter.sequence.status.seqActive;
   "Unit1.Em4.ControlNodes".cutter."step".transition[291] := ("Unit1.Em4.ControlNodes".cutter.sequence.status.currentStep = #JOB_2_STEP_91) AND "Unit1.Em4.ControlNodes".cutter.sequence.status.seqActive;
   #statTonTimer[291].TON(IN := ("Unit1.Em4.ControlNodes".cutter.sequence.status.currentStep = #JOB_2_STEP_91) AND "Unit1.Em4.ControlNodes".cutter.sequence.status.seqActive AND "Unit1.Em4.ControlNodes".cutter."step".transition[291],
                          PT := #SeqNoDelayTime);
   IF #statTonTimer[291].Q THEN
       "Unit1.Em4.ControlNodes".cutter.sequence.status.nextStep := #STEP_IDLE;
   END_IF;
END_REGION

REGION Network 17: *************** IMMEDIATE STOP ****************
END_REGION

REGION Network 18: Immediate Stop
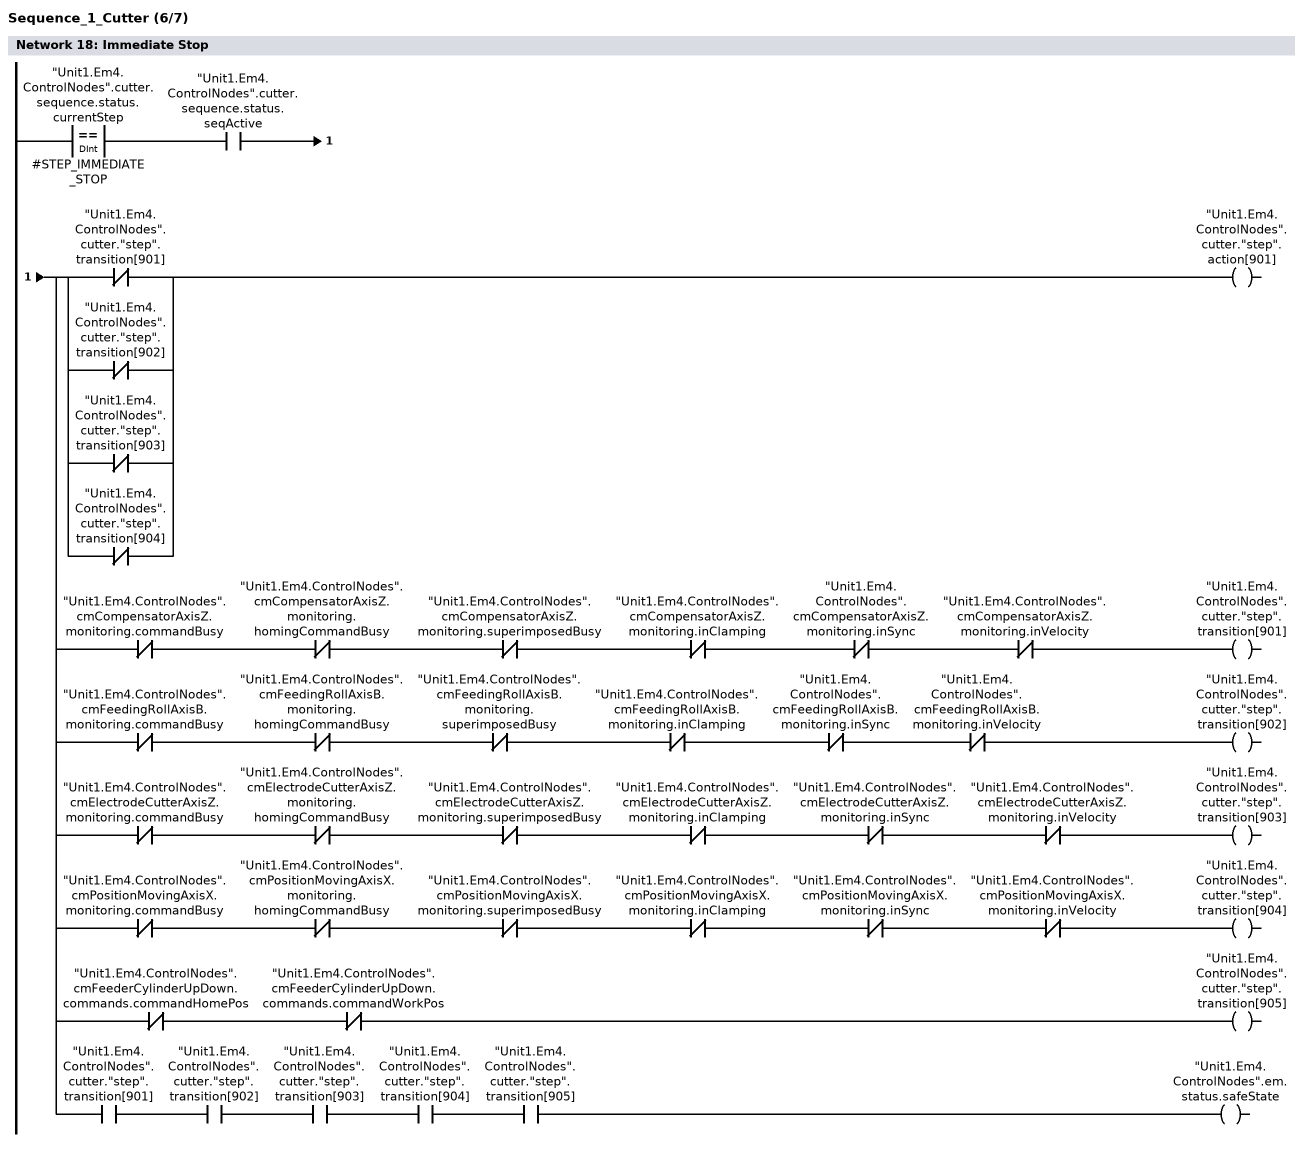
   RUNG wire#powerrail
      { S7_Templates := "SrcType := DInt" } EQ_Contact(in1 := "Unit1.Em4.ControlNodes".cutter.sequence.status.currentStep, in2 := #STEP_IMMEDIATE_STOP)
      Contact( "Unit1.Em4.ControlNodes".cutter.sequence.status.seqActive )
      wire#w1
      I_Contact( "Unit1.Em4.ControlNodes".cutter."step".transition[901] )
      wire#w2
      Coil( "Unit1.Em4.ControlNodes".cutter."step".action[901] )
   END_RUNG
   RUNG wire#w1
      I_Contact( "Unit1.Em4.ControlNodes".cutter."step".transition[902] )
   END_RUNG wire#w2
   RUNG wire#w1
      I_Contact( "Unit1.Em4.ControlNodes".cutter."step".transition[903] )
   END_RUNG wire#w2
   RUNG wire#w1
      I_Contact( "Unit1.Em4.ControlNodes".cutter."step".transition[904] )
   END_RUNG wire#w2
   RUNG wire#w1
      I_Contact( "Unit1.Em4.ControlNodes".cmCompensatorAxisZ.monitoring.commandBusy )
      I_Contact( "Unit1.Em4.ControlNodes".cmCompensatorAxisZ.monitoring.homingCommandBusy )
      I_Contact( "Unit1.Em4.ControlNodes".cmCompensatorAxisZ.monitoring.superimposedBusy )
      I_Contact( "Unit1.Em4.ControlNodes".cmCompensatorAxisZ.monitoring.inClamping )
      I_Contact( "Unit1.Em4.ControlNodes".cmCompensatorAxisZ.monitoring.inSync )
      I_Contact( "Unit1.Em4.ControlNodes".cmCompensatorAxisZ.monitoring.inVelocity )
      Coil( "Unit1.Em4.ControlNodes".cutter."step".transition[901] )
   END_RUNG
   RUNG wire#w1
      I_Contact( "Unit1.Em4.ControlNodes".cmFeedingRollAxisB.monitoring.commandBusy )
      I_Contact( "Unit1.Em4.ControlNodes".cmFeedingRollAxisB.monitoring.homingCommandBusy )
      I_Contact( "Unit1.Em4.ControlNodes".cmFeedingRollAxisB.monitoring.superimposedBusy )
      I_Contact( "Unit1.Em4.ControlNodes".cmFeedingRollAxisB.monitoring.inClamping )
      I_Contact( "Unit1.Em4.ControlNodes".cmFeedingRollAxisB.monitoring.inSync )
      I_Contact( "Unit1.Em4.ControlNodes".cmFeedingRollAxisB.monitoring.inVelocity )
      Coil( "Unit1.Em4.ControlNodes".cutter."step".transition[902] )
   END_RUNG
   RUNG wire#w1
      I_Contact( "Unit1.Em4.ControlNodes".cmElectrodeCutterAxisZ.monitoring.commandBusy )
      I_Contact( "Unit1.Em4.ControlNodes".cmElectrodeCutterAxisZ.monitoring.homingCommandBusy )
      I_Contact( "Unit1.Em4.ControlNodes".cmElectrodeCutterAxisZ.monitoring.superimposedBusy )
      I_Contact( "Unit1.Em4.ControlNodes".cmElectrodeCutterAxisZ.monitoring.inClamping )
      I_Contact( "Unit1.Em4.ControlNodes".cmElectrodeCutterAxisZ.monitoring.inSync )
      I_Contact( "Unit1.Em4.ControlNodes".cmElectrodeCutterAxisZ.monitoring.inVelocity )
      Coil( "Unit1.Em4.ControlNodes".cutter."step".transition[903] )
   END_RUNG
   RUNG wire#w1
      I_Contact( "Unit1.Em4.ControlNodes".cmPositionMovingAxisX.monitoring.commandBusy )
      I_Contact( "Unit1.Em4.ControlNodes".cmPositionMovingAxisX.monitoring.homingCommandBusy )
      I_Contact( "Unit1.Em4.ControlNodes".cmPositionMovingAxisX.monitoring.superimposedBusy )
      I_Contact( "Unit1.Em4.ControlNodes".cmPositionMovingAxisX.monitoring.inClamping )
      I_Contact( "Unit1.Em4.ControlNodes".cmPositionMovingAxisX.monitoring.inSync )
      I_Contact( "Unit1.Em4.ControlNodes".cmPositionMovingAxisX.monitoring.inVelocity )
      Coil( "Unit1.Em4.ControlNodes".cutter."step".transition[904] )
   END_RUNG
   RUNG wire#w1
      I_Contact( "Unit1.Em4.ControlNodes".cmFeederCylinderUpDown.commands.commandHomePos )
      I_Contact( "Unit1.Em4.ControlNodes".cmFeederCylinderUpDown.commands.commandWorkPos )
      Coil( "Unit1.Em4.ControlNodes".cutter."step".transition[905] )
   END_RUNG
   RUNG wire#w1
      Contact( "Unit1.Em4.ControlNodes".cutter."step".transition[901] )
      Contact( "Unit1.Em4.ControlNodes".cutter."step".transition[902] )
      Contact( "Unit1.Em4.ControlNodes".cutter."step".transition[903] )
      Contact( "Unit1.Em4.ControlNodes".cutter."step".transition[904] )
      Contact( "Unit1.Em4.ControlNodes".cutter."step".transition[905] )
      Coil( "Unit1.Em4.ControlNodes".em.status.safeState )
   END_RUNG
   // the same network as SCL:
   #_w1 := ("Unit1.Em4.ControlNodes".cutter.sequence.status.currentStep = #STEP_IMMEDIATE_STOP) AND "Unit1.Em4.ControlNodes".cutter.sequence.status.seqActive;
   "Unit1.Em4.ControlNodes".cutter."step".action[901] := #_w1 AND (NOT "Unit1.Em4.ControlNodes".cutter."step".transition[901] OR NOT "Unit1.Em4.ControlNodes".cutter."step".transition[902] OR NOT "Unit1.Em4.ControlNodes".cutter."step".transition[903] OR NOT "Unit1.Em4.ControlNodes".cutter."step".transition[904]);
   "Unit1.Em4.ControlNodes".cutter."step".transition[901] := #_w1 AND NOT "Unit1.Em4.ControlNodes".cmCompensatorAxisZ.monitoring.commandBusy AND NOT "Unit1.Em4.ControlNodes".cmCompensatorAxisZ.monitoring.homingCommandBusy AND NOT "Unit1.Em4.ControlNodes".cmCompensatorAxisZ.monitoring.superimposedBusy AND NOT "Unit1.Em4.ControlNodes".cmCompensatorAxisZ.monitoring.inClamping AND NOT "Unit1.Em4.ControlNodes".cmCompensatorAxisZ.monitoring.inSync AND NOT "Unit1.Em4.ControlNodes".cmCompensatorAxisZ.monitoring.inVelocity;
   "Unit1.Em4.ControlNodes".cutter."step".transition[902] := #_w1 AND NOT "Unit1.Em4.ControlNodes".cmFeedingRollAxisB.monitoring.commandBusy AND NOT "Unit1.Em4.ControlNodes".cmFeedingRollAxisB.monitoring.homingCommandBusy AND NOT "Unit1.Em4.ControlNodes".cmFeedingRollAxisB.monitoring.superimposedBusy AND NOT "Unit1.Em4.ControlNodes".cmFeedingRollAxisB.monitoring.inClamping AND NOT "Unit1.Em4.ControlNodes".cmFeedingRollAxisB.monitoring.inSync AND NOT "Unit1.Em4.ControlNodes".cmFeedingRollAxisB.monitoring.inVelocity;
   "Unit1.Em4.ControlNodes".cutter."step".transition[903] := #_w1 AND NOT "Unit1.Em4.ControlNodes".cmElectrodeCutterAxisZ.monitoring.commandBusy AND NOT "Unit1.Em4.ControlNodes".cmElectrodeCutterAxisZ.monitoring.homingCommandBusy AND NOT "Unit1.Em4.ControlNodes".cmElectrodeCutterAxisZ.monitoring.superimposedBusy AND NOT "Unit1.Em4.ControlNodes".cmElectrodeCutterAxisZ.monitoring.inClamping AND NOT "Unit1.Em4.ControlNodes".cmElectrodeCutterAxisZ.monitoring.inSync AND NOT "Unit1.Em4.ControlNodes".cmElectrodeCutterAxisZ.monitoring.inVelocity;
   "Unit1.Em4.ControlNodes".cutter."step".transition[904] := #_w1 AND NOT "Unit1.Em4.ControlNodes".cmPositionMovingAxisX.monitoring.commandBusy AND NOT "Unit1.Em4.ControlNodes".cmPositionMovingAxisX.monitoring.homingCommandBusy AND NOT "Unit1.Em4.ControlNodes".cmPositionMovingAxisX.monitoring.superimposedBusy AND NOT "Unit1.Em4.ControlNodes".cmPositionMovingAxisX.monitoring.inClamping AND NOT "Unit1.Em4.ControlNodes".cmPositionMovingAxisX.monitoring.inSync AND NOT "Unit1.Em4.ControlNodes".cmPositionMovingAxisX.monitoring.inVelocity;
   "Unit1.Em4.ControlNodes".cutter."step".transition[905] := #_w1 AND NOT "Unit1.Em4.ControlNodes".cmFeederCylinderUpDown.commands.commandHomePos AND NOT "Unit1.Em4.ControlNodes".cmFeederCylinderUpDown.commands.commandWorkPos;
   "Unit1.Em4.ControlNodes".em.status.safeState := #_w1 AND "Unit1.Em4.ControlNodes".cutter."step".transition[901] AND "Unit1.Em4.ControlNodes".cutter."step".transition[902] AND "Unit1.Em4.ControlNodes".cutter."step".transition[903] AND "Unit1.Em4.ControlNodes".cutter."step".transition[904] AND "Unit1.Em4.ControlNodes".cutter."step".transition[905];
END_REGION

REGION Network 19: *************** STATUS **********************
END_REGION

REGION Network 20: Sequence Status
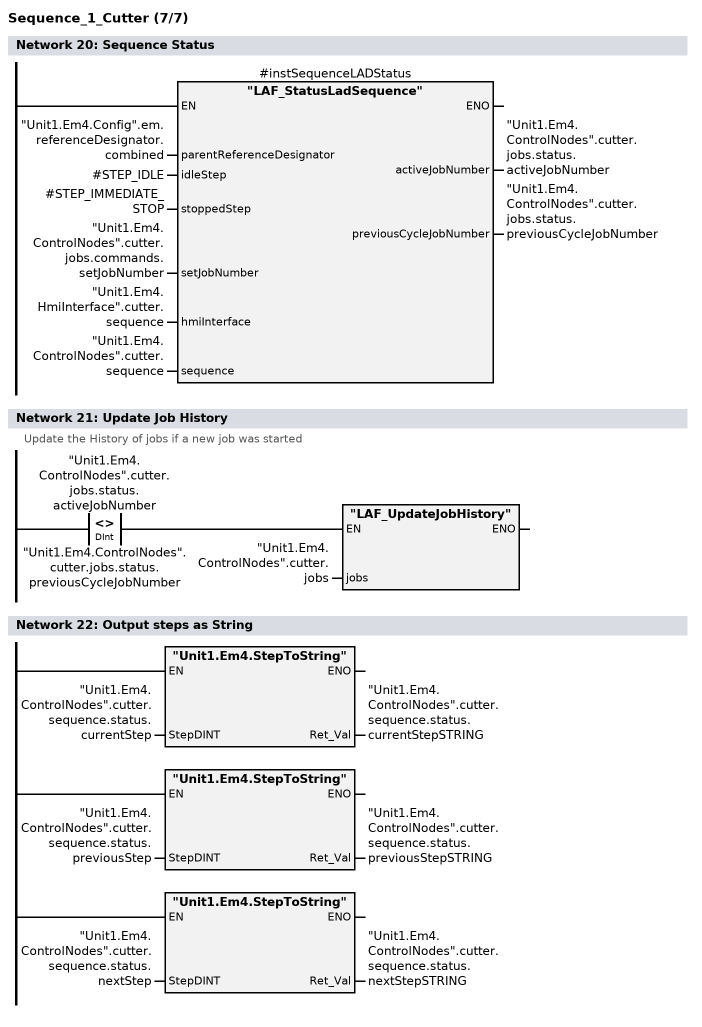
   RUNG wire#powerrail
      #instSequenceLADStatus(parentReferenceDesignator := "Unit1.Em4.Config".em.referenceDesignator.combined, idleStep := #STEP_IDLE, stoppedStep := #STEP_IMMEDIATE_STOP, setJobNumber := "Unit1.Em4.ControlNodes".cutter.jobs.commands.setJobNumber, hmiInterface := "Unit1.Em4.HmiInterface".cutter.sequence, sequence := "Unit1.Em4.ControlNodes".cutter.sequence, activeJobNumber => "Unit1.Em4.ControlNodes".cutter.jobs.status.activeJobNumber, previousCycleJobNumber => "Unit1.Em4.ControlNodes".cutter.jobs.status.previousCycleJobNumber)
   END_RUNG
   // the same network as SCL:
   #instSequenceLADStatus(parentReferenceDesignator := "Unit1.Em4.Config".em.referenceDesignator.combined,   // "LAF_StatusLadSequence"
                          idleStep := #STEP_IDLE,
                          stoppedStep := #STEP_IMMEDIATE_STOP,
                          setJobNumber := "Unit1.Em4.ControlNodes".cutter.jobs.commands.setJobNumber,
                          hmiInterface := "Unit1.Em4.HmiInterface".cutter.sequence,
                          sequence := "Unit1.Em4.ControlNodes".cutter.sequence,
                          activeJobNumber => "Unit1.Em4.ControlNodes".cutter.jobs.status.activeJobNumber,
                          previousCycleJobNumber => "Unit1.Em4.ControlNodes".cutter.jobs.status.previousCycleJobNumber);
END_REGION

REGION Network 21: Update Job History
   // Update the History of jobs if a new job was started
   RUNG wire#powerrail
      { S7_Templates := "SrcType := DInt" } NE_Contact(in1 := "Unit1.Em4.ControlNodes".cutter.jobs.status.activeJobNumber, in2 := "Unit1.Em4.ControlNodes".cutter.jobs.status.previousCycleJobNumber)
      "LAF_UpdateJobHistory"(jobs := "Unit1.Em4.ControlNodes".cutter.jobs)
   END_RUNG
   // the same network as SCL:
   IF "Unit1.Em4.ControlNodes".cutter.jobs.status.activeJobNumber <> "Unit1.Em4.ControlNodes".cutter.jobs.status.previousCycleJobNumber THEN
       "LAF_UpdateJobHistory"(jobs := "Unit1.Em4.ControlNodes".cutter.jobs);
   END_IF;
END_REGION

REGION Network 22: Output steps as String
   RUNG wire#powerrail
      "Unit1.Em4.StepToString"(StepDINT := "Unit1.Em4.ControlNodes".cutter.sequence.status.currentStep, Ret_Val => "Unit1.Em4.ControlNodes".cutter.sequence.status.currentStepSTRING)
   END_RUNG
   RUNG wire#powerrail
      "Unit1.Em4.StepToString"(StepDINT := "Unit1.Em4.ControlNodes".cutter.sequence.status.previousStep, Ret_Val => "Unit1.Em4.ControlNodes".cutter.sequence.status.previousStepSTRING)
   END_RUNG
   RUNG wire#powerrail
      "Unit1.Em4.StepToString"(StepDINT := "Unit1.Em4.ControlNodes".cutter.sequence.status.nextStep, Ret_Val => "Unit1.Em4.ControlNodes".cutter.sequence.status.nextStepSTRING)
   END_RUNG
   // the same network as SCL:
   "Unit1.Em4.ControlNodes".cutter.sequence.status.currentStepSTRING := "Unit1.Em4.StepToString"(StepDINT := "Unit1.Em4.ControlNodes".cutter.sequence.status.currentStep);
   "Unit1.Em4.ControlNodes".cutter.sequence.status.previousStepSTRING := "Unit1.Em4.StepToString"(StepDINT := "Unit1.Em4.ControlNodes".cutter.sequence.status.previousStep);
   "Unit1.Em4.ControlNodes".cutter.sequence.status.nextStepSTRING := "Unit1.Em4.StepToString"(StepDINT := "Unit1.Em4.ControlNodes".cutter.sequence.status.nextStep);
END_REGION
END_FUNCTION_BLOCK
